FUNCTION_BLOCK ConveyorLSC EXTENDS ConveyorSC
VAR_OUTPUT
	lifterError AT %I* : BOOL;
	
	extended AT %I* : BOOL;
	retracted AT %I* : BOOL;
END_VAR
VAR	
	lifterEnable AT %Q* : BOOL := TRUE;
	lifterDirection AT %Q* : BOOL; //FALSE = up, TRUE = down
	lifterPulse AT %Q* : BOOL;
	lifterReset AT %Q* : BOOL;
END_VAR
VAR	
	lifterMode : (HOLD, LIFTER_EXTEND, LIFTER_RETRACT); 
	lifterPulser : TP; //pulses are assumed to be low-high-low
END_VAR

SUPER^();

lifterOverride();

lifterSequence();

METHOD backward : BOOL
VAR_INPUT
END_VAR
END_METHOD

METHOD extend : BOOL
VAR_INPUT
END_VAR
lifterMode := LIFTER_EXTEND;
END_METHOD

METHOD forward : BOOL
VAR_INPUT
END_VAR
END_METHOD

METHOD PROTECTED lifterOverride : BOOL
VAR_INPUT
END_VAR
IF
	(extended AND lifterMode = LIFTER_EXTEND) OR
	(retracted AND lifterMode = LIFTER_RETRACT)
THEN
	lifterMode := HOLD;
END_IF
END_METHOD

METHOD PROTECTED lifterSequence : BOOL
VAR_INPUT
END_VAR
VAR
	nextOp, prevOp : INT;
END_VAR
lifterPulser(IN:= , PT:= pulseWidth, Q=> , ET=> );
lifterPulser.IN := 
	lifterEnable AND 
	NOT lifterError AND 
	NOT lifterReset AND 
	( (lifterMode = LIFTER_EXTEND AND NOT extended) OR (lifterMode = LIFTER_RETRACT AND NOT retracted) ) AND
	lifterPulser.Q; //self-ending pulse

lifterPulse := lifterPulser.Q AND lifterPulser.ET < pulseWidth/2;
END_METHOD

METHOD reset : BOOL
VAR_INPUT
END_VAR
position := 0;
velocity := velocity; //no change

extend();
END_METHOD

METHOD retract : BOOL
VAR_INPUT
END_VAR
lifterMode := LIFTER_RETRACT;
END_METHOD

END_FUNCTION_BLOCK

(* stored: Version 1.1.0.1, ProductVersion 3.1.4024.11
   POU ConveyorLSC: Id {4f6cfb6d-6de1-4268-b14b-f837abcc174e}, SpecialFunc None
   Folder Private: Id {2dd6dc1f-1fb9-40a8-bfe0-bcc4441b187c}
   Folder Properties: Id {662df990-c299-470b-a18e-00f0d61ccba1}
   Folder Unused: Id {bec3ed47-90ed-4528-8dd6-b850ab70f8f2}
   Method backward: Id {c19450f5-569e-456f-87af-46b285416a87}
   Method extend: Id {134a21db-f191-4efc-8030-b5c51776b21e}
   Method forward: Id {b50396ae-3747-4bf2-a6cd-af89c8af7dd2}
   Method lifterOverride: Id {e01b1a57-c0ed-4e15-a5d5-b6d037837ced}
   Method lifterSequence: Id {3151b70e-86df-4eac-bfc8-17c901b97fc9}
   Method reset: Id {ebbae814-1c37-427f-a836-796c3bf16516}
   Method retract: Id {e3aaa3fe-86c4-448a-a6b0-436a4b77fc00} *)
